Staubli VAL3: cmdEnableOp.pgx

public program cmdEnableOp(num x_nAxNum)
begin
  //设置'Enable Operation'
  if bOpeEnabled[x_nAxNum]==false
    doFaultReset[x_nAxNum]=false
    doSwitchOn[x_nAxNum]=false
    doEnableOp[x_nAxNum]=false
    doEnableVoltage[x_nAxNum]=true
    doQuickStop[x_nAxNum]=true
    delay(0.1)
    doSwitchOn[x_nAxNum]=true
    delay(0.1)
    doEnableOp[x_nAxNum]=true
    delay(0.1)
  endIf
end
